(* Logix 5000 project; controller DispersionPlc vendor 1 type 14 code 108 rev 34.11; software revision 34.01; part 9 of 22 *)
(* tags used below, declared in another part *)
   ONS : BOOL[32];
   B4320_HighHighLevel : BOOL;
   B4320_HighHighLevelMessage : BOOL;
   B4320_LastTrasferredLb : REAL;
   B4320_PumpAutoCommand : BOOL;
   B4320_PumpManStart : AOI_Toggle;
   B4320_Selected : BOOL;
   B4320_SelectPB : BOOL;
   B4320_TransferStarted : BOOL;
   BLANK64 : Stp64;
   CurrentTrasferredLb : REAL;
   Drum_Addition_K400 : Seq64;
   Drum_Addition_T430X : Seq64;
   Drum_Addition_T430X_Timer : TIMER;
   Drum_Addition_Timer : TIMER;
   Drum_Transfer : BOOL;
   Estop_Inx : ALIAS FOR Local:3:I.Data.3;
   FIT_S47_1 : AStd_AnalogInput;
   FIT_S47_1_AOI : AStd_AI_AOI;
   FIT_S47_1MassFlowLBMin : REAL;
   FIT_S47_1PulseCounter : COUNTER;
   FlowmeterPulse : BOOL;
   HMI_Drum_Addition_T430X_Timer : REAL;
   HMI_Drum_Addition_Timer : REAL;
   HMI_Mon_Isolation_K400_Timer : REAL;
   INX_Alarm : BOOL[32];
   INX_AlarmTmr : TIMER[32];
   Mon_Destination_K400 : BOOL;
   Mon_Destination_K400_ONS : BOOL;
   Mon_Destination_K400_PB : BOOL;
   Mon_Destination_T4301 : BOOL;
   Mon_Destination_T4301_ONS : BOOL;
   Mon_Destination_T4301_PB : BOOL;
   Mon_Isolation_K400_Timer : TIMER;
   Mon_Purge_Transfer_K400 : Seq64;
   Mon_Purge_Transfer_T430X : Seq64;
   Mon_Tank_Destination : DINT;
   MON_VALV_ENBL : DINT;
   MON_VALV_ENBL_BIT1 : BOOL;
   MON_VALV_ENBL_PB1 : BOOL;
   MONOMER_RESET : BOOL;
   NM_4303_AOI : AStd_AI_AOI;
   NM_4303_O2 : AStd_AnalogInput;
   NM_4303_O2_SIGNAL : REAL;
   One_Shots : DINT;
   PIDE_TCV_S47_1_AutoSP : REAL;
   PulseBit : INT;
   PulseToLbFactor : REAL;
   S47_HighHighLevel : BOOL;
   S47_HighHighLevelMessage : BOOL;
   S47_HighLevel : BOOL;
   S47_LastTrasferredLb : REAL;
   S47_OkToRun : BOOL;
   S47_PumpAutoCommand : BOOL;
   S47_PumpIsRunning : BOOL;
   S47_PumpManCommand : BOOL;
   S47_PumpManStartPB : BOOL;
   S47_PumpManStopPB : BOOL;
   S47_Selected : BOOL;
   S47_SelectPB : BOOL;
   S47_Toggle : AOI_Toggle;
   S47_transfer_amount : REAL;
   S47_TransferLimit : REAL;
   S47_transferLimitMessage : BOOL;
   S47_TransferSetpoint : REAL;
   S47_TransferStarted : BOOL;
   S47_TransferStartPB : BOOL;
   S47_TransferStopPB : BOOL;
   ST_K400_1 : REAL;
   StorageBit : INT;
   SV_4303_01 : ALIAS FOR Local:5:O.Data.8;
   SV_4303_03 : BOOL;
   SV_4303_03_Enable_PB : BOOL;
   SV_4303_04 : BOOL;
   SV_4303_04_Enable_PB : BOOL;
   Tank47_Level : INT;
   Tank_Destination_ONS : BOOL;
   Task_Permissive : DINT[2];
   TCV_S47_1_AutoCommand : REAL;
   TCV_S47_1_AutoManTransition : BOOL;
   TCV_S47_1_AutoManTransitionDelay : TIMER;
   TCV_S47_1_AutoPB : BOOL;
   TCV_S47_1_AutoSelected : BOOL;
   TCV_S47_1_Command : REAL;
   TCV_S47_1_ManAutoTransition : BOOL;
   TCV_S47_1_ManAutoTransitionDelay : TIMER;
   TCV_S47_1_ManualCommand : DINT;
   TCV_S47_1_ManualPB : BOOL;
   TCV_S47_1_ManualSelected : BOOL;
   TCV_S47_1Output : Analog_Scale;
   TIT_S47_1 : AStd_AnalogInput;
   TIT_S47_1_AOI : AStd_AI_AOI;
   TIT_S47_1_HiHi : REAL;
   TOGGLE : BOOL;
   TRANS_PUMP_P_4320_RUN : ALIAS FOR Local:1:O.Data[0].6;
   TransferDone : BOOL;
   TransferOffset : REAL;
   TransferSetpoint : REAL;
   TransferStopValueLb : REAL;
   W4303_Pump : VFD;
   XV_4303_03 : BOOL;
   XV_4303_04 : BOOL;
   XV_4303_05 : BOOL;
   XV_K400_03_SEQCLOSE : BOOL;
   XV_K400_03_SEQOPEN : BOOL;
   XV_S47_1_CloseCommand : BOOL;
   XV_S47_1_IsClosed : BOOL;
   XV_S47_2_CloseCommand : BOOL;
   XV_S47_2_IsClosed : BOOL;
   XV_S47_2_IsOpen : BOOL;
   XV_S47_2_OpenCommand : BOOL;
   ZSC_4303_03 : BOOL;
   ZSC_4303_04 : BOOL;
   ZSC_4303_1 : ALIAS FOR Local:2:I.Data.7;
   ZSC_K400_03 : BOOL;
   ZSO_4303_03 : BOOL;
   ZSO_4303_04 : BOOL;
   ZSO_4303_05 : BOOL;
   ZSO_4303_1 : ALIAS FOR Local:2:I.Data.6;
   ZSO_K400_03 : BOOL;
(* MainProgram, continued *)

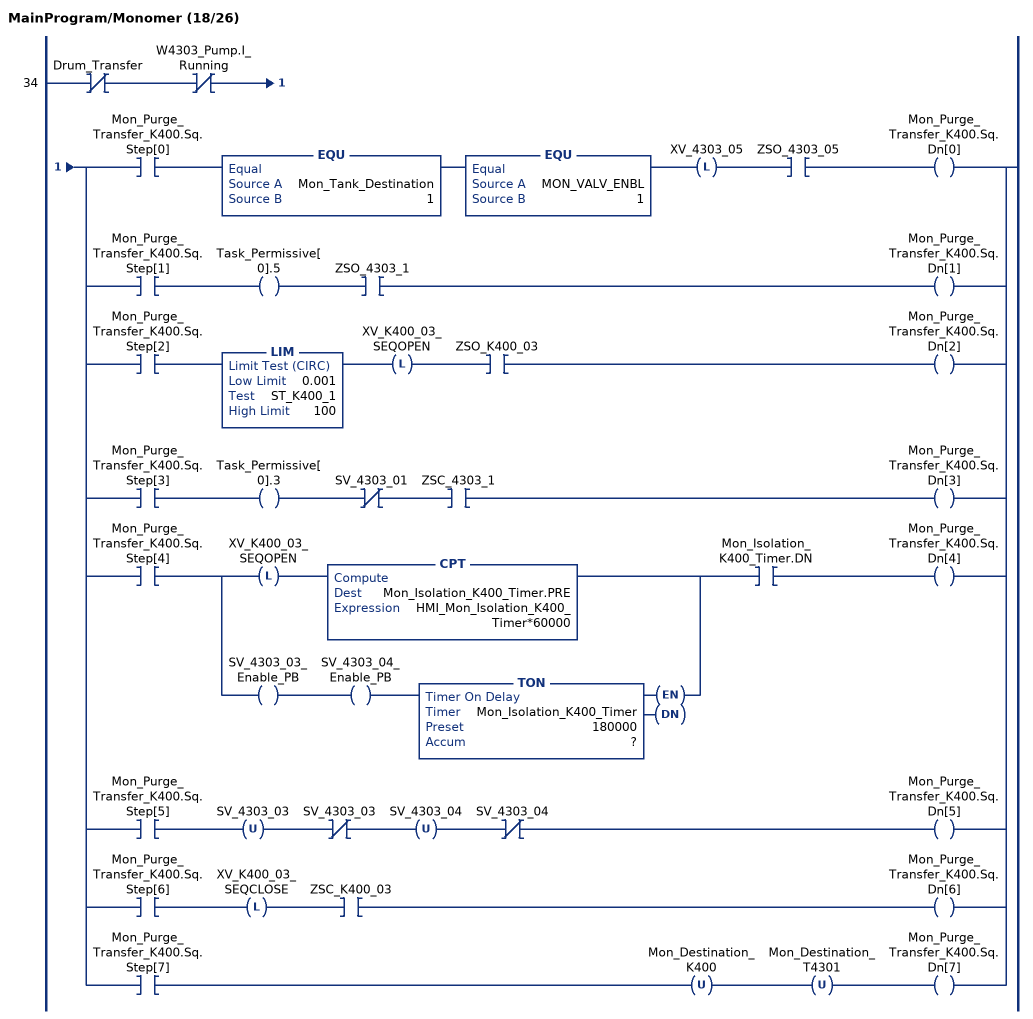
   [picture p157: MainProgram/Monomer rungs 34-34]
   34: XIO(Drum_Transfer)XIO(W4303_Pump.I_Running)[XIC(Mon_Purge_Transfer_K400.Sq.Step[0]) EQU(Mon_Tank_Destination,1) EQU(MON_VALV_ENBL,1) OTL(XV_4303_05) XIC(ZSO_4303_05) OTE(Mon_Purge_Transfer_K400.Sq.Dn[0]) ,XIC(Mon_Purge_Transfer_K400.Sq.Step[1]) OTE(Task_Permissive[0].5) XIC(ZSO_4303_1) OTE(Mon_Purge_Transfer_K400.Sq.Dn[1]) ,XIC(Mon_Purge_Transfer_K400.Sq.Step[2]) LIM(0.001,ST_K400_1,100) OTL(XV_K400_03_SEQOPEN) XIC(ZSO_K400_03) OTE(Mon_Purge_Transfer_K400.Sq.Dn[2]) ,XIC(Mon_Purge_Transfer_K400.Sq.Step[3]) OTE(Task_Permissive[0].3) XIO(SV_4303_01) XIC(ZSC_4303_1) OTE(Mon_Purge_Transfer_K400.Sq.Dn[3]) ,XIC(Mon_Purge_Transfer_K400.Sq.Step[4]) [OTL(XV_K400_03_SEQOPEN) CPT(Mon_Isolation_K400_Timer.PRE,HMI_Mon_Isolation_K400_Timer*60000) ,OTE(SV_4303_03_Enable_PB) OTE(SV_4303_04_Enable_PB) TON(Mon_Isolation_K400_Timer,?,?) ] XIC(Mon_Isolation_K400_Timer.DN) OTE(Mon_Purge_Transfer_K400.Sq.Dn[4]) ,XIC(Mon_Purge_Transfer_K400.Sq.Step[5]) OTU(SV_4303_03) XIO(SV_4303_03) OTU(SV_4303_04) XIO(SV_4303_04) OTE(Mon_Purge_Transfer_K400.Sq.Dn[5]) ,XIC(Mon_Purge_Transfer_K400.Sq.Step[6]) OTL(XV_K400_03_SEQCLOSE) XIC(ZSC_K400_03) OTE(Mon_Purge_Transfer_K400.Sq.Dn[6]) ,XIC(Mon_Purge_Transfer_K400.Sq.Step[7]) OTU(Mon_Destination_K400) OTU(Mon_Destination_T4301) OTE(Mon_Purge_Transfer_K400.Sq.Dn[7]) ];
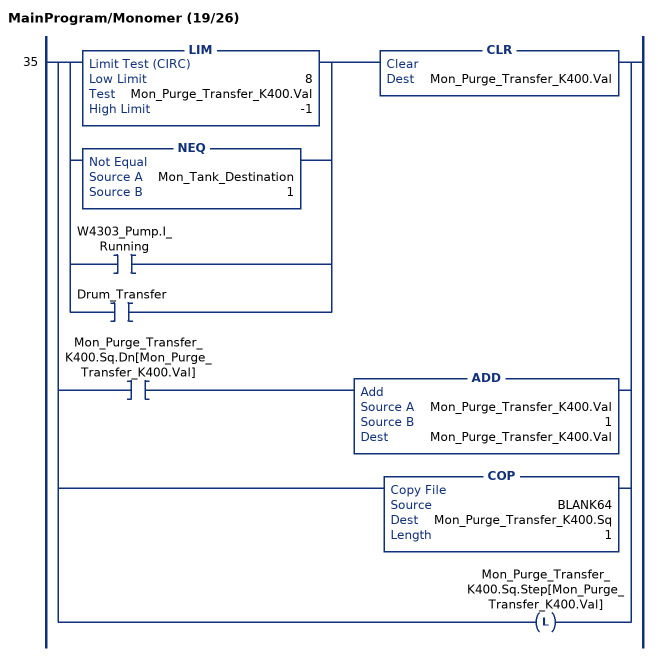
   35: [[LIM(8,Mon_Purge_Transfer_K400.Val,-1) ,NEQ(Mon_Tank_Destination,1) ,XIC(W4303_Pump.I_Running) ,XIC(Drum_Transfer) ] CLR(Mon_Purge_Transfer_K400.Val) ,XIC(Mon_Purge_Transfer_K400.Sq.Dn[Mon_Purge_Transfer_K400.Val]) ADD(Mon_Purge_Transfer_K400.Val,1,Mon_Purge_Transfer_K400.Val) ,COP(BLANK64,Mon_Purge_Transfer_K400.Sq,1) ,OTL(Mon_Purge_Transfer_K400.Sq.Step[Mon_Purge_Transfer_K400.Val]) ];
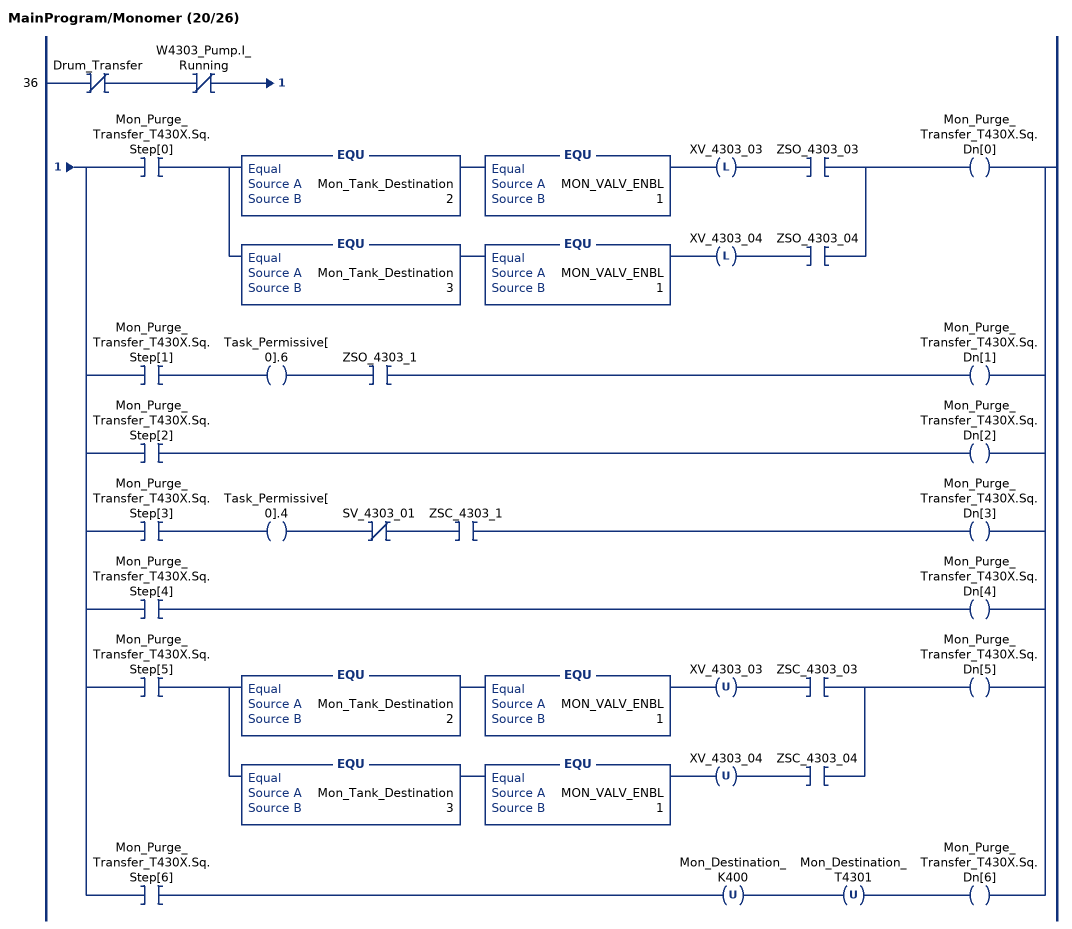
   36: XIO(Drum_Transfer)XIO(W4303_Pump.I_Running)[XIC(Mon_Purge_Transfer_T430X.Sq.Step[0]) [EQU(Mon_Tank_Destination,2) EQU(MON_VALV_ENBL,1) OTL(XV_4303_03) XIC(ZSO_4303_03) ,EQU(Mon_Tank_Destination,3) EQU(MON_VALV_ENBL,1) OTL(XV_4303_04) XIC(ZSO_4303_04) ] OTE(Mon_Purge_Transfer_T430X.Sq.Dn[0]) ,XIC(Mon_Purge_Transfer_T430X.Sq.Step[1]) OTE(Task_Permissive[0].6) XIC(ZSO_4303_1) OTE(Mon_Purge_Transfer_T430X.Sq.Dn[1]) ,XIC(Mon_Purge_Transfer_T430X.Sq.Step[2]) OTE(Mon_Purge_Transfer_T430X.Sq.Dn[2]) ,XIC(Mon_Purge_Transfer_T430X.Sq.Step[3]) OTE(Task_Permissive[0].4) XIO(SV_4303_01) XIC(ZSC_4303_1) OTE(Mon_Purge_Transfer_T430X.Sq.Dn[3]) ,XIC(Mon_Purge_Transfer_T430X.Sq.Step[4]) OTE(Mon_Purge_Transfer_T430X.Sq.Dn[4]) ,XIC(Mon_Purge_Transfer_T430X.Sq.Step[5]) [EQU(Mon_Tank_Destination,2) EQU(MON_VALV_ENBL,1) OTU(XV_4303_03) XIC(ZSC_4303_03) ,EQU(Mon_Tank_Destination,3) EQU(MON_VALV_ENBL,1) OTU(XV_4303_04) XIC(ZSC_4303_04) ] OTE(Mon_Purge_Transfer_T430X.Sq.Dn[5]) ,XIC(Mon_Purge_Transfer_T430X.Sq.Step[6]) OTU(Mon_Destination_K400) OTU(Mon_Destination_T4301) OTE(Mon_Purge_Transfer_T430X.Sq.Dn[6]) ];
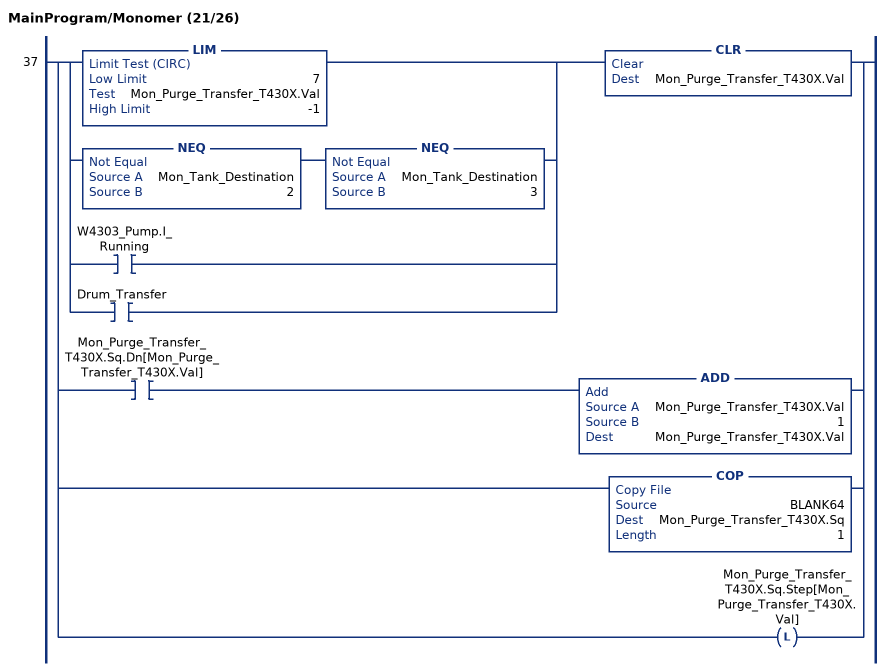
   37: [[LIM(7,Mon_Purge_Transfer_T430X.Val,-1) ,NEQ(Mon_Tank_Destination,2) NEQ(Mon_Tank_Destination,3) ,XIC(W4303_Pump.I_Running) ,XIC(Drum_Transfer) ] CLR(Mon_Purge_Transfer_T430X.Val) ,XIC(Mon_Purge_Transfer_T430X.Sq.Dn[Mon_Purge_Transfer_T430X.Val]) ADD(Mon_Purge_Transfer_T430X.Val,1,Mon_Purge_Transfer_T430X.Val) ,COP(BLANK64,Mon_Purge_Transfer_T430X.Sq,1) ,OTL(Mon_Purge_Transfer_T430X.Sq.Step[Mon_Purge_Transfer_T430X.Val]) ];
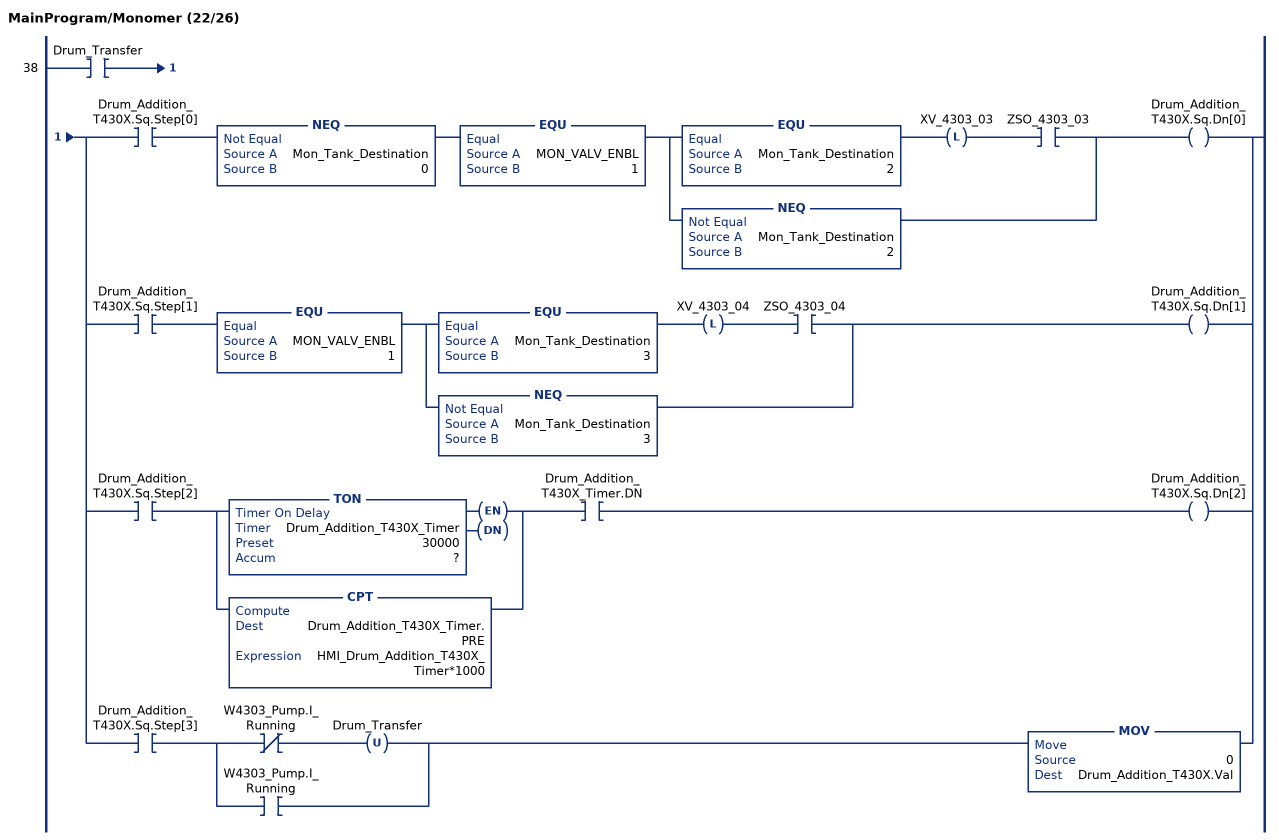
   38: XIC(Drum_Transfer)[XIC(Drum_Addition_T430X.Sq.Step[0]) NEQ(Mon_Tank_Destination,0) EQU(MON_VALV_ENBL,1) [EQU(Mon_Tank_Destination,2) OTL(XV_4303_03) XIC(ZSO_4303_03) ,NEQ(Mon_Tank_Destination,2) ] OTE(Drum_Addition_T430X.Sq.Dn[0]) ,XIC(Drum_Addition_T430X.Sq.Step[1]) EQU(MON_VALV_ENBL,1) [EQU(Mon_Tank_Destination,3) OTL(XV_4303_04) XIC(ZSO_4303_04) ,NEQ(Mon_Tank_Destination,3) ] OTE(Drum_Addition_T430X.Sq.Dn[1]) ,XIC(Drum_Addition_T430X.Sq.Step[2]) [TON(Drum_Addition_T430X_Timer,?,?) ,CPT(Drum_Addition_T430X_Timer.PRE,HMI_Drum_Addition_T430X_Timer*1000) ] XIC(Drum_Addition_T430X_Timer.DN) OTE(Drum_Addition_T430X.Sq.Dn[2]) ,XIC(Drum_Addition_T430X.Sq.Step[3]) [XIO(W4303_Pump.I_Running) OTU(Drum_Transfer) ,XIC(W4303_Pump.I_Running) ] MOV(0,Drum_Addition_T430X.Val) ];
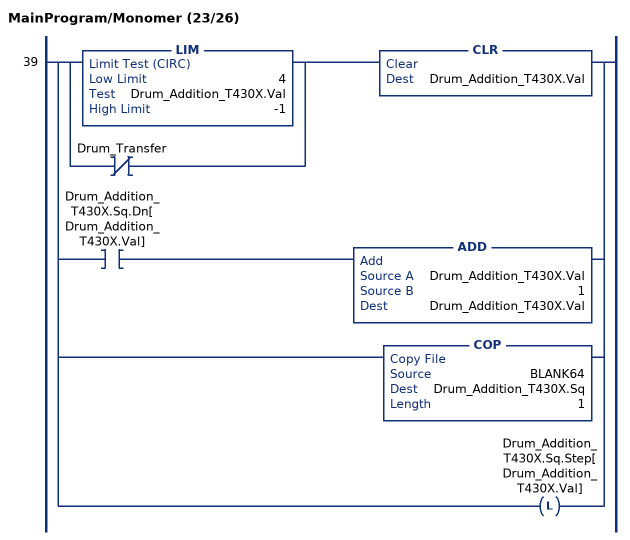
   39: [[LIM(4,Drum_Addition_T430X.Val,-1) ,XIO(Drum_Transfer) ] CLR(Drum_Addition_T430X.Val) ,XIC(Drum_Addition_T430X.Sq.Dn[Drum_Addition_T430X.Val]) ADD(Drum_Addition_T430X.Val,1,Drum_Addition_T430X.Val) ,COP(BLANK64,Drum_Addition_T430X.Sq,1) ,OTL(Drum_Addition_T430X.Sq.Step[Drum_Addition_T430X.Val]) ];
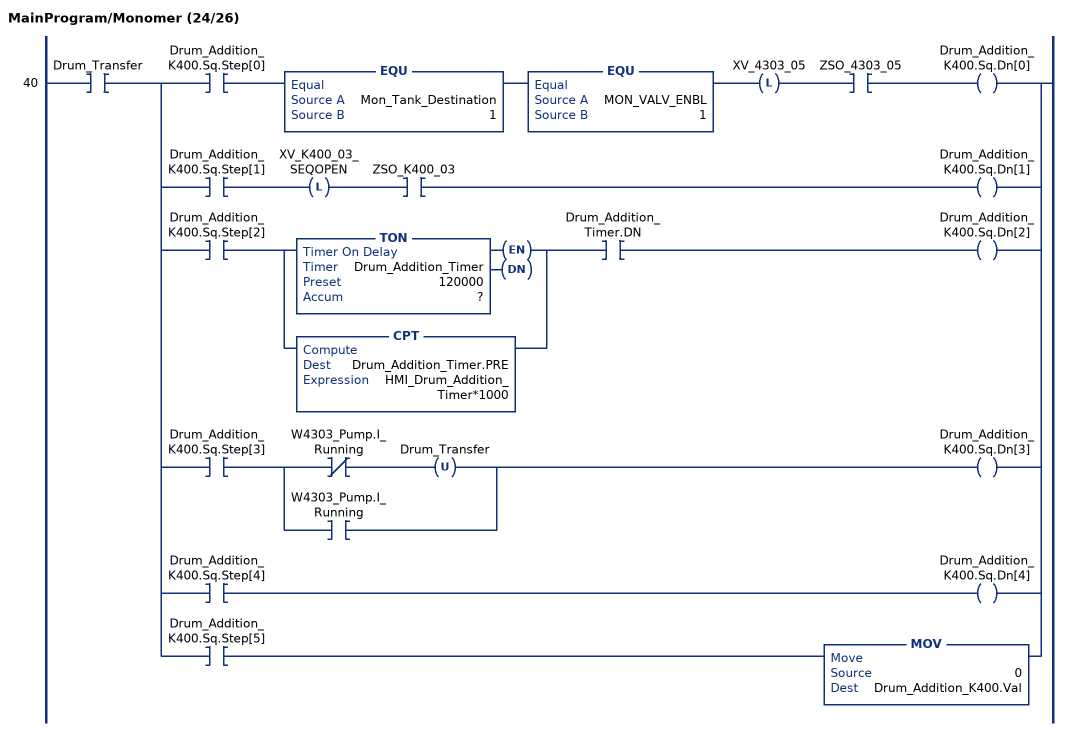
   40: XIC(Drum_Transfer)[XIC(Drum_Addition_K400.Sq.Step[0]) EQU(Mon_Tank_Destination,1) EQU(MON_VALV_ENBL,1) OTL(XV_4303_05) XIC(ZSO_4303_05) OTE(Drum_Addition_K400.Sq.Dn[0]) ,XIC(Drum_Addition_K400.Sq.Step[1]) OTL(XV_K400_03_SEQOPEN) XIC(ZSO_K400_03) OTE(Drum_Addition_K400.Sq.Dn[1]) ,XIC(Drum_Addition_K400.Sq.Step[2]) [TON(Drum_Addition_Timer,?,?) ,CPT(Drum_Addition_Timer.PRE,HMI_Drum_Addition_Timer*1000) ] XIC(Drum_Addition_Timer.DN) OTE(Drum_Addition_K400.Sq.Dn[2]) ,XIC(Drum_Addition_K400.Sq.Step[3]) [XIO(W4303_Pump.I_Running) OTU(Drum_Transfer) ,XIC(W4303_Pump.I_Running) ] OTE(Drum_Addition_K400.Sq.Dn[3]) ,XIC(Drum_Addition_K400.Sq.Step[4]) OTE(Drum_Addition_K400.Sq.Dn[4]) ,XIC(Drum_Addition_K400.Sq.Step[5]) MOV(0,Drum_Addition_K400.Val) ];
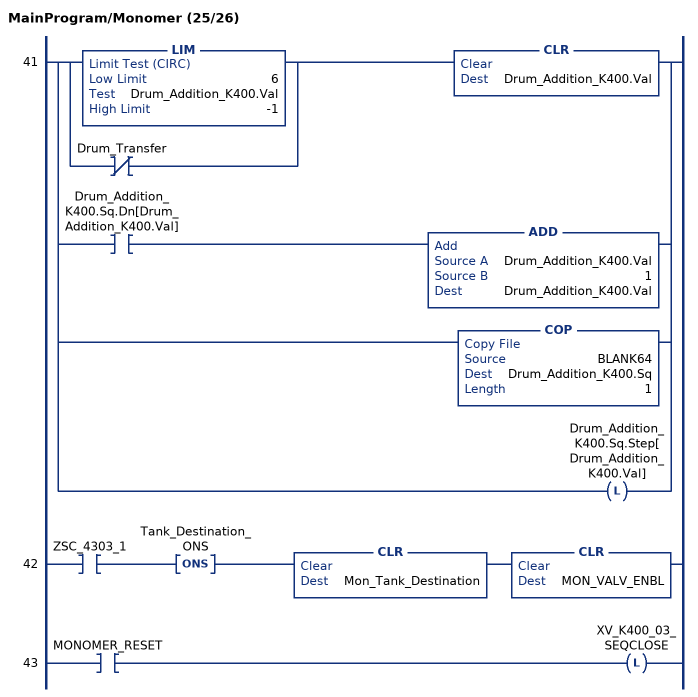
   41: [[LIM(6,Drum_Addition_K400.Val,-1) ,XIO(Drum_Transfer) ] CLR(Drum_Addition_K400.Val) ,XIC(Drum_Addition_K400.Sq.Dn[Drum_Addition_K400.Val]) ADD(Drum_Addition_K400.Val,1,Drum_Addition_K400.Val) ,COP(BLANK64,Drum_Addition_K400.Sq,1) ,OTL(Drum_Addition_K400.Sq.Step[Drum_Addition_K400.Val]) ];
   42: XIC(ZSC_4303_1)ONS(Tank_Destination_ONS)CLR(Mon_Tank_Destination)CLR(MON_VALV_ENBL);
   43: XIC(MONOMER_RESET)OTL(XV_K400_03_SEQCLOSE);
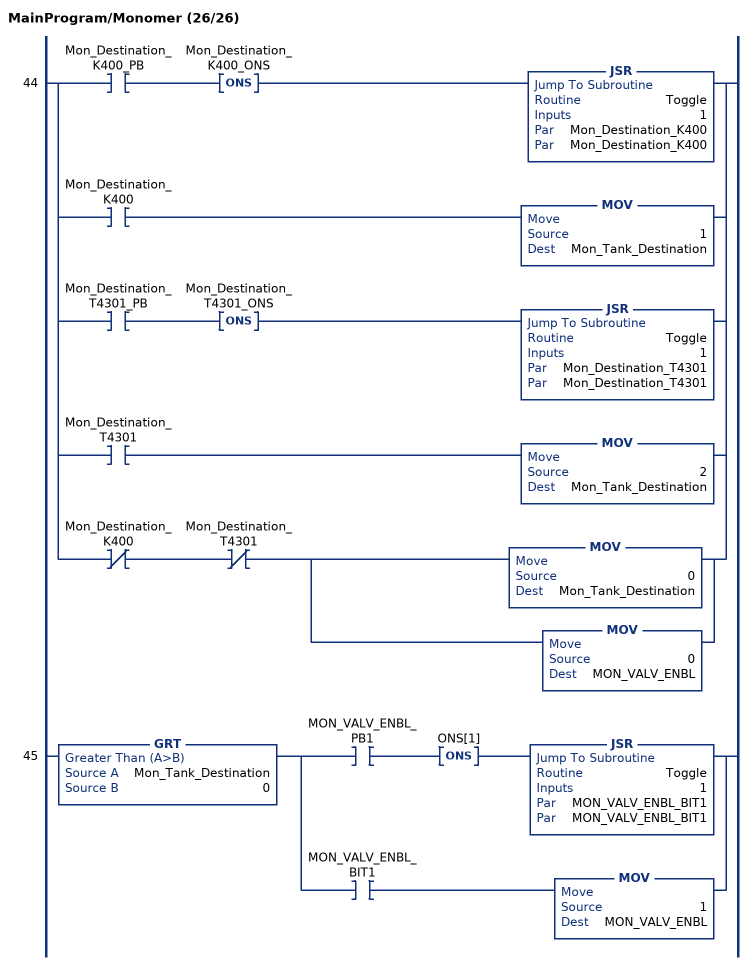
   44: [[XIC(Mon_Destination_K400_PB) ONS(Mon_Destination_K400_ONS) JSR(Toggle,1,Mon_Destination_K400,Mon_Destination_K400) ,XIC(Mon_Destination_K400) MOV(1,Mon_Tank_Destination) ] ,[XIC(Mon_Destination_T4301_PB) ONS(Mon_Destination_T4301_ONS) JSR(Toggle,1,Mon_Destination_T4301,Mon_Destination_T4301) ,XIC(Mon_Destination_T4301) MOV(2,Mon_Tank_Destination) ] ,XIO(Mon_Destination_K400) XIO(Mon_Destination_T4301) [MOV(0,Mon_Tank_Destination) ,MOV(0,MON_VALV_ENBL) ] ];
   45: GRT(Mon_Tank_Destination,0)[XIC(MON_VALV_ENBL_PB1) ONS(ONS[1]) JSR(Toggle,1,MON_VALV_ENBL_BIT1,MON_VALV_ENBL_BIT1) ,XIC(MON_VALV_ENBL_BIT1) MOV(1,MON_VALV_ENBL) ];
END_ROUTINE

ROUTINE NM4303   (* ladder *)
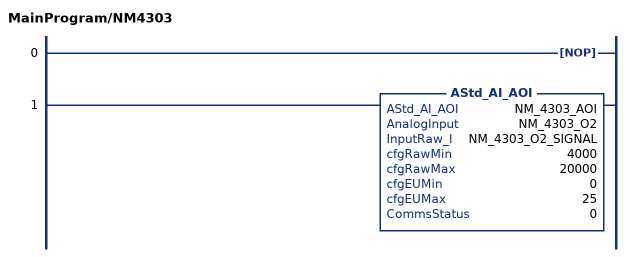
   0: NOP();
   1: AStd_AI_AOI(NM_4303_AOI,NM_4303_O2,NM_4303_O2_SIGNAL,4000,20000,0,25,0);
END_ROUTINE

ROUTINE S47_Transfer   (* ladder *)
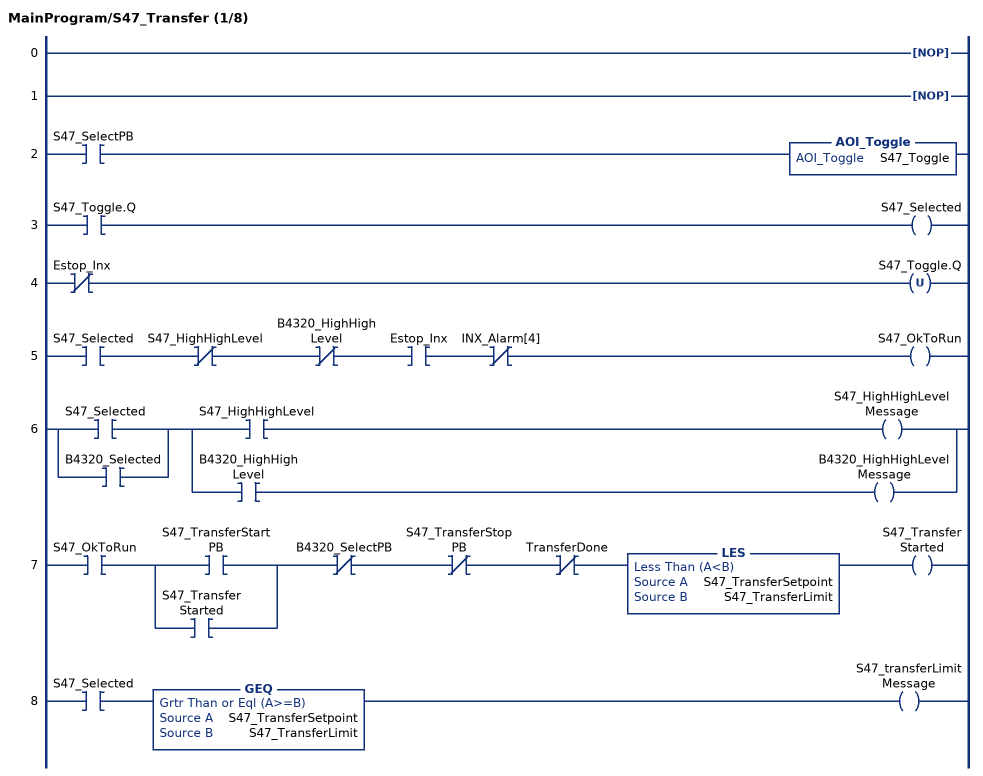
   0: NOP();
   1: NOP();
   2: XIC(S47_SelectPB)AOI_Toggle(S47_Toggle);
   3: XIC(S47_Toggle.Q)OTE(S47_Selected);
   4: XIO(Estop_Inx)OTU(S47_Toggle.Q);
   5: XIC(S47_Selected)XIO(S47_HighHighLevel)XIO(B4320_HighHighLevel)XIC(Estop_Inx)XIO(INX_Alarm[4])OTE(S47_OkToRun);
   6: [XIC(S47_Selected) ,XIC(B4320_Selected) ][XIC(S47_HighHighLevel) OTE(S47_HighHighLevelMessage) ,XIC(B4320_HighHighLevel) OTE(B4320_HighHighLevelMessage) ];
   7: XIC(S47_OkToRun)[XIC(S47_TransferStartPB) ,XIC(S47_TransferStarted) ]XIO(B4320_SelectPB)XIO(S47_TransferStopPB)XIO(TransferDone)LES(S47_TransferSetpoint,S47_TransferLimit)OTE(S47_TransferStarted);
   8: XIC(S47_Selected)GEQ(S47_TransferSetpoint,S47_TransferLimit)OTE(S47_transferLimitMessage);
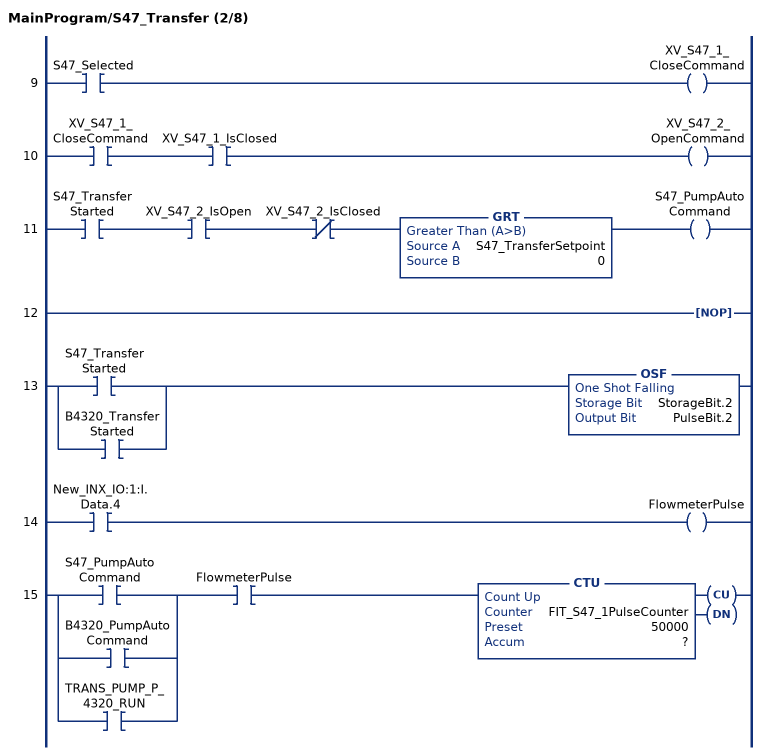
   9: XIC(S47_Selected)OTE(XV_S47_1_CloseCommand);
   10: XIC(XV_S47_1_CloseCommand)XIC(XV_S47_1_IsClosed)OTE(XV_S47_2_OpenCommand);
   11: XIC(S47_TransferStarted)XIC(XV_S47_2_IsOpen)XIO(XV_S47_2_IsClosed)GRT(S47_TransferSetpoint,0)OTE(S47_PumpAutoCommand);
   12: NOP();
   13: [XIC(S47_TransferStarted) ,XIC(B4320_TransferStarted) ]OSF(StorageBit.2,PulseBit.2);
   14: XIC(New_INX_IO:1:I.Data.4)OTE(FlowmeterPulse);
   15: [XIC(S47_PumpAutoCommand) ,XIC(B4320_PumpAutoCommand) ,XIC(TRANS_PUMP_P_4320_RUN) ]XIC(FlowmeterPulse)CTU(FIT_S47_1PulseCounter,?,?);
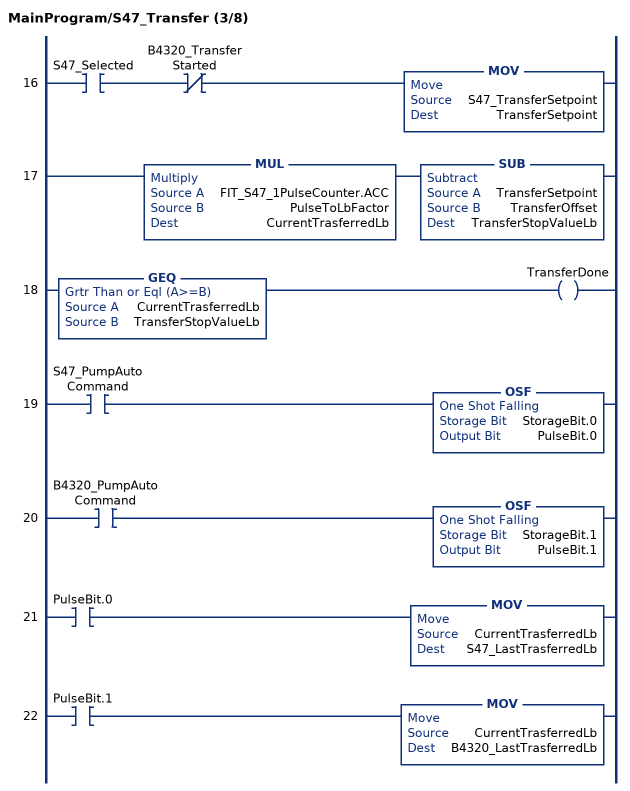
   16: XIC(S47_Selected)XIO(B4320_TransferStarted)MOV(S47_TransferSetpoint,TransferSetpoint);
   17: MUL(FIT_S47_1PulseCounter.ACC,PulseToLbFactor,CurrentTrasferredLb)SUB(TransferSetpoint,TransferOffset,TransferStopValueLb);
   18: GEQ(CurrentTrasferredLb,TransferStopValueLb)OTE(TransferDone);
   19: XIC(S47_PumpAutoCommand)OSF(StorageBit.0,PulseBit.0);
   20: XIC(B4320_PumpAutoCommand)OSF(StorageBit.1,PulseBit.1);
   21: XIC(PulseBit.0)MOV(CurrentTrasferredLb,S47_LastTrasferredLb);
   22: XIC(PulseBit.1)MOV(CurrentTrasferredLb,B4320_LastTrasferredLb);
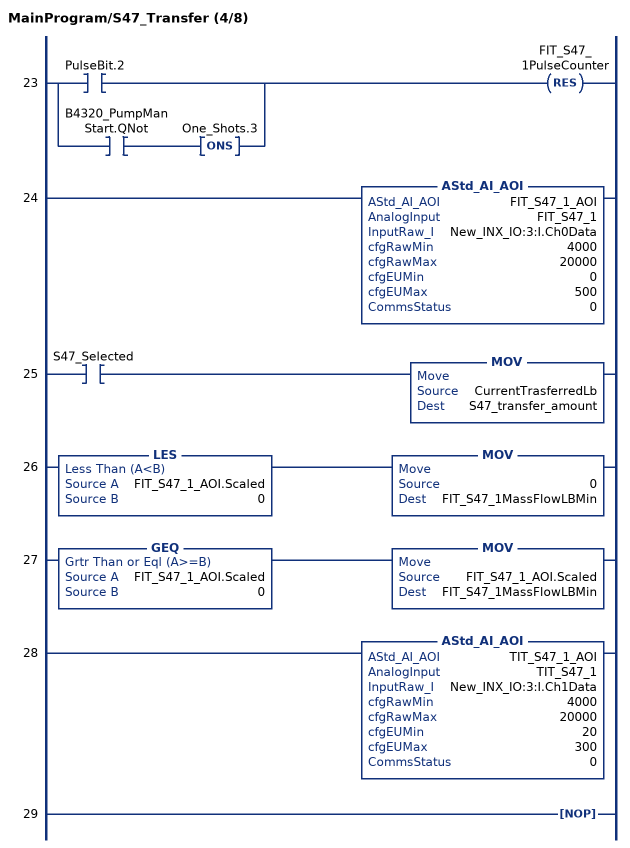
   23: [XIC(PulseBit.2) ,XIC(B4320_PumpManStart.QNot) ONS(One_Shots.3) ]RES(FIT_S47_1PulseCounter);
   24: AStd_AI_AOI(FIT_S47_1_AOI,FIT_S47_1,New_INX_IO:3:I.Ch0Data,4000,20000,0,500,0);
   25: XIC(S47_Selected)MOV(CurrentTrasferredLb,S47_transfer_amount);
   26: LES(FIT_S47_1_AOI.Scaled,0)MOV(0,FIT_S47_1MassFlowLBMin);
   27: GEQ(FIT_S47_1_AOI.Scaled,0)MOV(FIT_S47_1_AOI.Scaled,FIT_S47_1MassFlowLBMin);
   28: AStd_AI_AOI(TIT_S47_1_AOI,TIT_S47_1,New_INX_IO:3:I.Ch1Data,4000,20000,20,300,0);
   29: NOP();
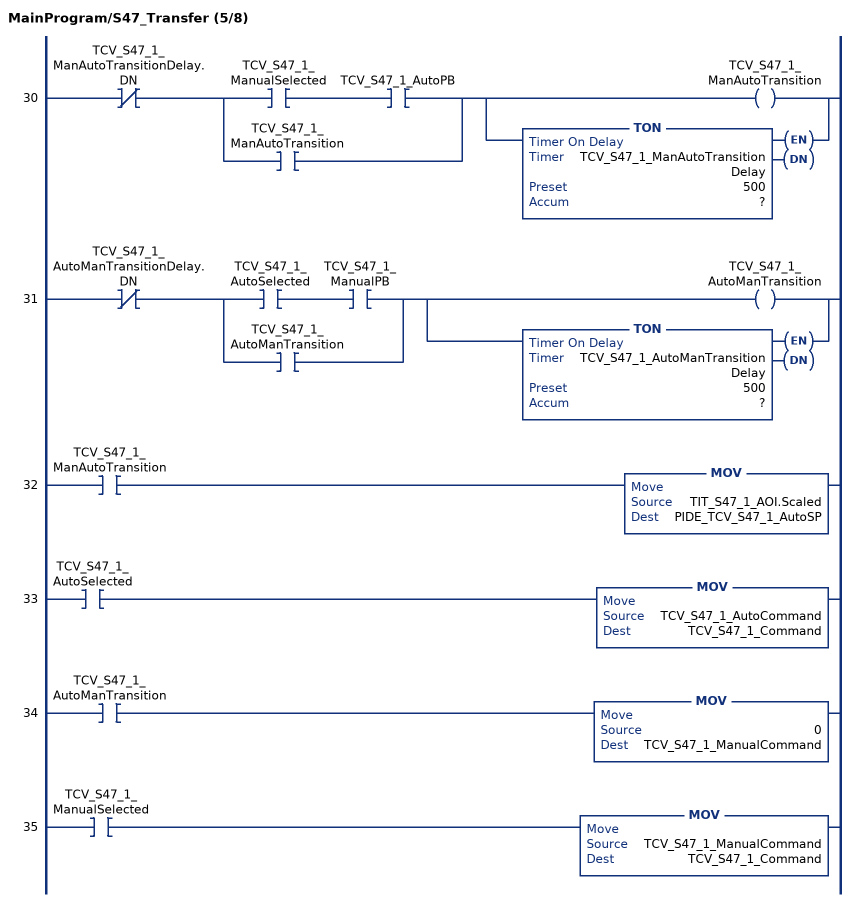
   30: XIO(TCV_S47_1_ManAutoTransitionDelay.DN)[XIC(TCV_S47_1_ManualSelected) XIC(TCV_S47_1_AutoPB) ,XIC(TCV_S47_1_ManAutoTransition) ][OTE(TCV_S47_1_ManAutoTransition) ,TON(TCV_S47_1_ManAutoTransitionDelay,?,?) ];
   31: XIO(TCV_S47_1_AutoManTransitionDelay.DN)[XIC(TCV_S47_1_AutoSelected) XIC(TCV_S47_1_ManualPB) ,XIC(TCV_S47_1_AutoManTransition) ][OTE(TCV_S47_1_AutoManTransition) ,TON(TCV_S47_1_AutoManTransitionDelay,?,?) ];
   32: XIC(TCV_S47_1_ManAutoTransition)MOV(TIT_S47_1_AOI.Scaled,PIDE_TCV_S47_1_AutoSP);
   33: XIC(TCV_S47_1_AutoSelected)MOV(TCV_S47_1_AutoCommand,TCV_S47_1_Command);
   34: XIC(TCV_S47_1_AutoManTransition)MOV(0,TCV_S47_1_ManualCommand);
   35: XIC(TCV_S47_1_ManualSelected)MOV(TCV_S47_1_ManualCommand,TCV_S47_1_Command);
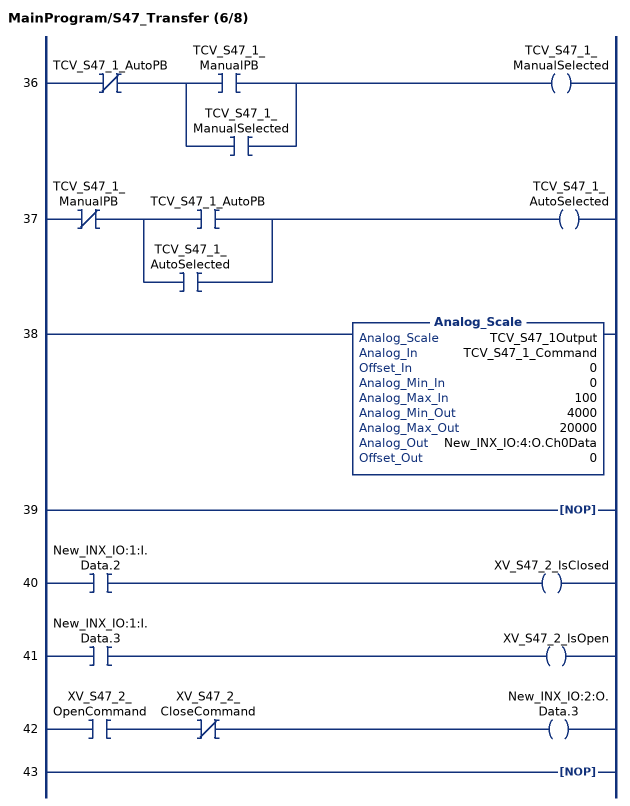
   36: XIO(TCV_S47_1_AutoPB)[XIC(TCV_S47_1_ManualPB) ,XIC(TCV_S47_1_ManualSelected) ]OTE(TCV_S47_1_ManualSelected);
   37: XIO(TCV_S47_1_ManualPB)[XIC(TCV_S47_1_AutoPB) ,XIC(TCV_S47_1_AutoSelected) ]OTE(TCV_S47_1_AutoSelected);
   38: Analog_Scale(TCV_S47_1Output,TCV_S47_1_Command,0,0,100,4000,20000,New_INX_IO:4:O.Ch0Data,0);
   39: NOP();
   40: XIC(New_INX_IO:1:I.Data.2)OTE(XV_S47_2_IsClosed);
   41: XIC(New_INX_IO:1:I.Data.3)OTE(XV_S47_2_IsOpen);
   42: XIC(XV_S47_2_OpenCommand)XIO(XV_S47_2_CloseCommand)OTE(New_INX_IO:2:O.Data.3);
   43: NOP();
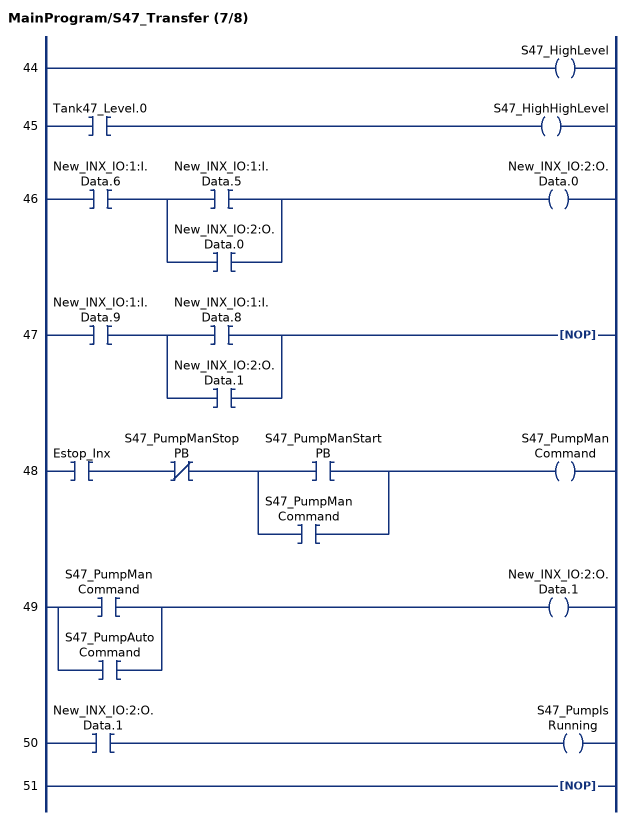
   44: OTE(S47_HighLevel);
   45: XIC(Tank47_Level.0)OTE(S47_HighHighLevel);
   46: XIC(New_INX_IO:1:I.Data.6)[XIC(New_INX_IO:1:I.Data.5) ,XIC(New_INX_IO:2:O.Data.0) ]OTE(New_INX_IO:2:O.Data.0);
   47: XIC(New_INX_IO:1:I.Data.9)[XIC(New_INX_IO:1:I.Data.8) ,XIC(New_INX_IO:2:O.Data.1) ]NOP();
   48: XIC(Estop_Inx)XIO(S47_PumpManStopPB)[XIC(S47_PumpManStartPB) ,XIC(S47_PumpManCommand) ]OTE(S47_PumpManCommand);
   49: [XIC(S47_PumpManCommand) ,XIC(S47_PumpAutoCommand) ]OTE(New_INX_IO:2:O.Data.1);
   50: XIC(New_INX_IO:2:O.Data.1)OTE(S47_PumpIsRunning);
   51: NOP();
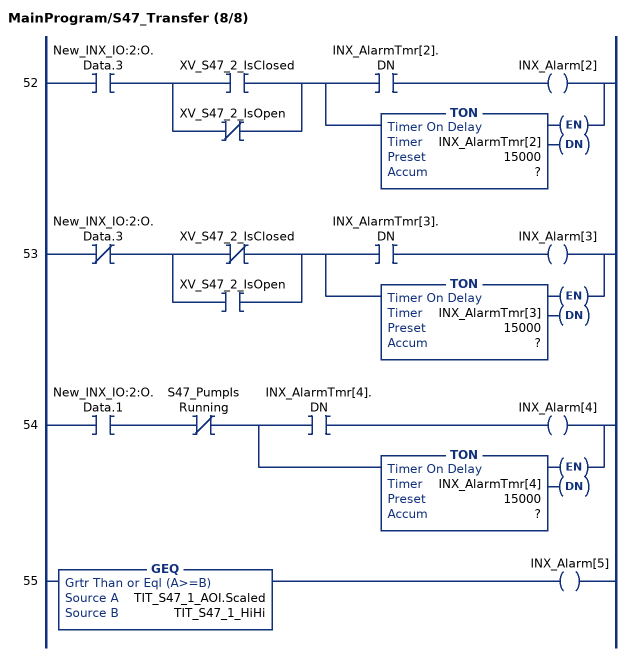
   52: XIC(New_INX_IO:2:O.Data.3)[XIC(XV_S47_2_IsClosed) ,XIO(XV_S47_2_IsOpen) ][XIC(INX_AlarmTmr[2].DN) OTE(INX_Alarm[2]) ,TON(INX_AlarmTmr[2],?,?) ];
   53: XIO(New_INX_IO:2:O.Data.3)[XIO(XV_S47_2_IsClosed) ,XIC(XV_S47_2_IsOpen) ][XIC(INX_AlarmTmr[3].DN) OTE(INX_Alarm[3]) ,TON(INX_AlarmTmr[3],?,?) ];
   54: XIC(New_INX_IO:2:O.Data.1)XIO(S47_PumpIsRunning)[XIC(INX_AlarmTmr[4].DN) OTE(INX_Alarm[4]) ,TON(INX_AlarmTmr[4],?,?) ];
   55: GEQ(TIT_S47_1_AOI.Scaled,TIT_S47_1_HiHi)OTE(INX_Alarm[5]);
END_ROUTINE
